// TIA Portal V17 export
// export: Created 2024-08-20T13:26:07.0461176Z, ExportSetting WithDefaults, DisplayName Totally Integrated Automation Portal, DisplayVersion V17 Update 4, DisplayName TIA Portal Openness, DisplayVersion V17 Update 4, DisplayName TIA Portal Version Control Interface, DisplayVersion V17, DisplayName STEP 7 Professional, DisplayVersion V17 Update 4, DisplayName STEP 7 Safety, DisplayVersion V17, DisplayName WinCC Advanced, DisplayVersion V17 Update 4
FUNCTION "MB-03" : Void   // FC24, LAD
TITLE = Lógica de acionamento do motor
{ S7_Optimized_Access := 'FALSE' }
VERSION : 0.1
// stored: AutoNumber false, IsIECCheckEnabled false, SetENOAutomatically false, UDAEnableTagReadback false
   VAR_TEMP
      IM : Bool;   // Intertravamento manual = 0
      IA : Bool;   // Intertravamento automáticol = 0
      HABM : Bool;   // Habilita funcionamento manual = 1
      HABA : Bool;   // Habilita funcionamento automático = 1
      CLM : Bool;   // Comando liga motor
      PROT : Bool;   // Proteção do motor acionada
   END_VAR
BEGIN

REGION Network 1: Intertravamento maual/automático
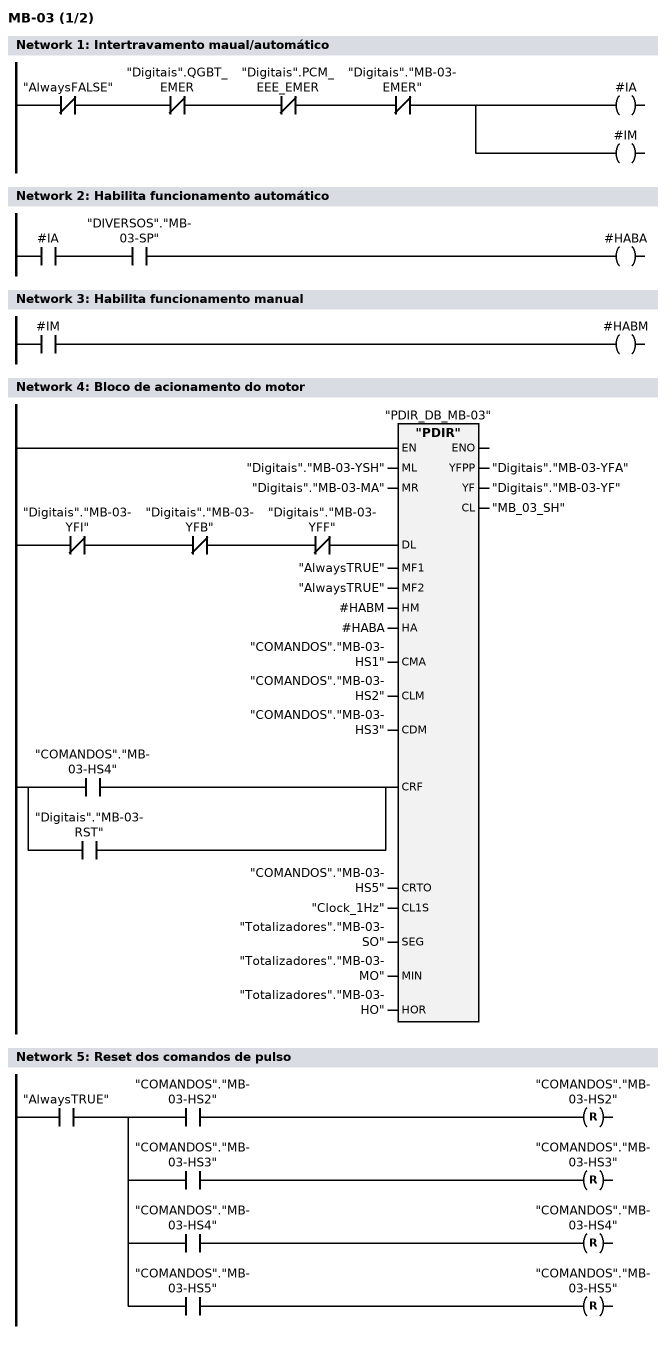
   RUNG wire#powerrail
      I_Contact( "AlwaysFALSE" )
      I_Contact( "Digitais".QGBT_EMER )
      I_Contact( "Digitais".PCM_EEE_EMER )
      I_Contact( "Digitais"."MB-03-EMER" )
      wire#w1
      Coil( #IA )
   END_RUNG
   RUNG wire#w1
      Coil( #IM )
   END_RUNG
   // the same network as SCL:
   #IA := NOT "AlwaysFALSE" AND NOT "Digitais".QGBT_EMER AND NOT "Digitais".PCM_EEE_EMER AND NOT "Digitais"."MB-03-EMER";
   #IM := #IA;
END_REGION

REGION Network 2: Habilita funcionamento automático
   RUNG wire#powerrail
      Contact( #IA )
      Contact( "DIVERSOS"."MB-03-SP" )
      Coil( #HABA )
   END_RUNG
   // the same network as SCL:
   #HABA := #IA AND "DIVERSOS"."MB-03-SP";
END_REGION

REGION Network 3: Habilita funcionamento manual
   RUNG wire#powerrail
      Contact( #IM )
      Coil( #HABM )
   END_RUNG
   // the same network as SCL:
   #HABM := #IM;
END_REGION

REGION Network 4: Bloco de acionamento do motor
   RUNG wire#powerrail
      "PDIR_DB_MB-03"(DL := wire#w1, CRF := wire#w2, ML := "Digitais"."MB-03-YSH", MR := "Digitais"."MB-03-MA", MF1 := "AlwaysTRUE", MF2 := "AlwaysTRUE", HM := #HABM, HA := #HABA, CMA := "COMANDOS"."MB-03-HS1", CLM := "COMANDOS"."MB-03-HS2", CDM := "COMANDOS"."MB-03-HS3", CRTO := "COMANDOS"."MB-03-HS5", CL1S := "Clock_1Hz", SEG := "Totalizadores"."MB-03-SO", MIN := "Totalizadores"."MB-03-MO", HOR := "Totalizadores"."MB-03-HO", YFPP => "Digitais"."MB-03-YFA", YF => "Digitais"."MB-03-YF", CL => "MB_03_SH")
   END_RUNG
   RUNG wire#powerrail
      I_Contact( "Digitais"."MB-03-YFI" )
      I_Contact( "Digitais"."MB-03-YFB" )
      I_Contact( "Digitais"."MB-03-YFF" )
   END_RUNG wire#w1
   RUNG wire#powerrail
      Contact( "COMANDOS"."MB-03-HS4" )
   END_RUNG wire#w2
   RUNG wire#powerrail
      Contact( "Digitais"."MB-03-RST" )
   END_RUNG wire#w2
   // the same network as SCL:
   "PDIR_DB_MB-03"(ML := "Digitais"."MB-03-YSH",   // "PDIR"
                   MR := "Digitais"."MB-03-MA",
                   DL := NOT "Digitais"."MB-03-YFI" AND NOT "Digitais"."MB-03-YFB" AND NOT "Digitais"."MB-03-YFF",
                   MF1 := "AlwaysTRUE",
                   MF2 := "AlwaysTRUE",
                   HM := #HABM,
                   HA := #HABA,
                   CMA := "COMANDOS"."MB-03-HS1",
                   CLM := "COMANDOS"."MB-03-HS2",
                   CDM := "COMANDOS"."MB-03-HS3",
                   CRF := "COMANDOS"."MB-03-HS4" OR "Digitais"."MB-03-RST",
                   CRTO := "COMANDOS"."MB-03-HS5",
                   CL1S := "Clock_1Hz",
                   SEG := "Totalizadores"."MB-03-SO",
                   MIN := "Totalizadores"."MB-03-MO",
                   HOR := "Totalizadores"."MB-03-HO",
                   YFPP => "Digitais"."MB-03-YFA",
                   YF => "Digitais"."MB-03-YF",
                   CL => "MB_03_SH");
END_REGION

REGION Network 5: Reset dos comandos de pulso
   RUNG wire#powerrail
      Contact( "AlwaysTRUE" )
      wire#w1
      Contact( "COMANDOS"."MB-03-HS2" )
      R_Coil( "COMANDOS"."MB-03-HS2" )
   END_RUNG
   RUNG wire#w1
      Contact( "COMANDOS"."MB-03-HS3" )
      R_Coil( "COMANDOS"."MB-03-HS3" )
   END_RUNG
   RUNG wire#w1
      Contact( "COMANDOS"."MB-03-HS4" )
      R_Coil( "COMANDOS"."MB-03-HS4" )
   END_RUNG
   RUNG wire#w1
      Contact( "COMANDOS"."MB-03-HS5" )
      R_Coil( "COMANDOS"."MB-03-HS5" )
   END_RUNG
   // the same network as SCL:
   IF "AlwaysTRUE" AND "COMANDOS"."MB-03-HS2" THEN "COMANDOS"."MB-03-HS2" := FALSE; END_IF;
   IF "AlwaysTRUE" AND "COMANDOS"."MB-03-HS3" THEN "COMANDOS"."MB-03-HS3" := FALSE; END_IF;
   IF "AlwaysTRUE" AND "COMANDOS"."MB-03-HS4" THEN "COMANDOS"."MB-03-HS4" := FALSE; END_IF;
   IF "AlwaysTRUE" AND "COMANDOS"."MB-03-HS5" THEN "COMANDOS"."MB-03-HS5" := FALSE; END_IF;
END_REGION

REGION Network 6: Elevatoria principal modo automatico
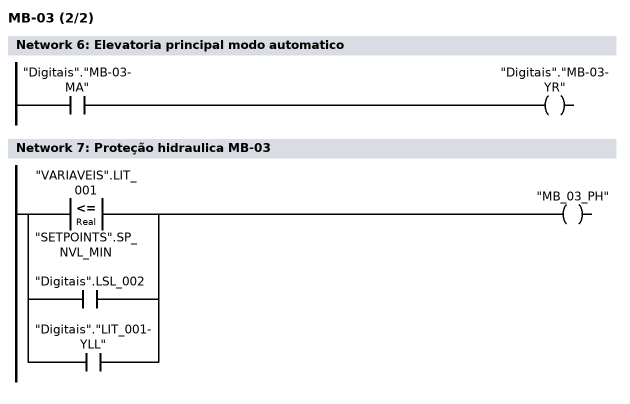
   RUNG wire#powerrail
      Contact( "Digitais"."MB-03-MA" )
      Coil( "Digitais"."MB-03-YR" )
   END_RUNG
   // the same network as SCL:
   "Digitais"."MB-03-YR" := "Digitais"."MB-03-MA";
END_REGION

REGION Network 7: Proteção hidraulica MB-03
   RUNG wire#powerrail
      { S7_Templates := "SrcType := Real" } LE_Contact(in1 := "VARIAVEIS".LIT_001, in2 := "SETPOINTS".SP_NVL_MIN)
      wire#w1
      Coil( "MB_03_PH" )
   END_RUNG
   RUNG wire#powerrail
      Contact( "Digitais".LSL_002 )
   END_RUNG wire#w1
   RUNG wire#powerrail
      Contact( "Digitais"."LIT_001-YLL" )
   END_RUNG wire#w1
   // the same network as SCL:
   "MB_03_PH" := ("VARIAVEIS".LIT_001 <= "SETPOINTS".SP_NVL_MIN) OR "Digitais".LSL_002 OR "Digitais"."LIT_001-YLL";
END_REGION
END_FUNCTION
